TYPE J1939_outputs :
STRUCT
	TxCounter : UINT;
	RxCounter   : UINT;
	NoOfTxMessages    : UINT;
	TxMessage  : ARRAY [0..1] OF VARTYPE_EXTCANQUEUE;
END_STRUCT
END_TYPE

(* stored: Version 1.1.0.1, ProductVersion 3.1.4024.9
   DUT J1939_outputs: Id {9288d42f-473b-49cb-b515-f2f8f634e386} *)
